  965 = 'Mc_Warnings Default 965' | German: 'Mc_Warnings German 965' | French: 'Mc_Warnings French 965'
  966 = 'Mc_Warnings Default 966' | German: 'Mc_Warnings German 966' | French: 'Mc_Warnings French 966'
  967 = 'Mc_Warnings Default 967' | German: 'Mc_Warnings German 967' | French: 'Mc_Warnings French 967'
  968 = 'Mc_Warnings Default 968' | German: 'Mc_Warnings German 968' | French: 'Mc_Warnings French 968'
  969 = 'Mc_Warnings Default 969' | German: 'Mc_Warnings German 969' | French: 'Mc_Warnings French 969'
  970 = 'Mc_Warnings Default 970' | German: 'Mc_Warnings German 970' | French: 'Mc_Warnings French 970'
  971 = 'Mc_Warnings Default 971' | German: 'Mc_Warnings German 971' | French: 'Mc_Warnings French 971'
  972 = 'Mc_Warnings Default 972' | German: 'Mc_Warnings German 972' | French: 'Mc_Warnings French 972'
  973 = 'Mc_Warnings Default 973' | German: 'Mc_Warnings German 973' | French: 'Mc_Warnings French 973'
  974 = 'Mc_Warnings Default 974' | German: 'Mc_Warnings German 974' | French: 'Mc_Warnings French 974'
  975 = 'Mc_Warnings Default 975' | German: 'Mc_Warnings German 975' | French: 'Mc_Warnings French 975'
  976 = 'Mc_Warnings Default 976' | German: 'Mc_Warnings German 976' | French: 'Mc_Warnings French 976'
  977 = 'Mc_Warnings Default 977' | German: 'Mc_Warnings German 977' | French: 'Mc_Warnings French 977'
  978 = 'Mc_Warnings Default 978' | German: 'Mc_Warnings German 978' | French: 'Mc_Warnings French 978'
  979 = 'Mc_Warnings Default 979' | German: 'Mc_Warnings German 979' | French: 'Mc_Warnings French 979'
  980 = 'Mc_Warnings Default 980' | German: 'Mc_Warnings German 980' | French: 'Mc_Warnings French 980'
  981 = 'Mc_Warnings Default 981' | German: 'Mc_Warnings German 981' | French: 'Mc_Warnings French 981'
  982 = 'Mc_Warnings Default 982' | German: 'Mc_Warnings German 982' | French: 'Mc_Warnings French 982'
  983 = 'Mc_Warnings Default 983' | German: 'Mc_Warnings German 983' | French: 'Mc_Warnings French 983'
  984 = 'Mc_Warnings Default 984' | German: 'Mc_Warnings German 984' | French: 'Mc_Warnings French 984'
  985 = 'Mc_Warnings Default 985' | German: 'Mc_Warnings German 985' | French: 'Mc_Warnings French 985'
  986 = 'Mc_Warnings Default 986' | German: 'Mc_Warnings German 986' | French: 'Mc_Warnings French 986'
  987 = 'Mc_Warnings Default 987' | German: 'Mc_Warnings German 987' | French: 'Mc_Warnings French 987'
  988 = 'Mc_Warnings Default 988' | German: 'Mc_Warnings German 988' | French: 'Mc_Warnings French 988'
  989 = 'Mc_Warnings Default 989' | German: 'Mc_Warnings German 989' | French: 'Mc_Warnings French 989'
  990 = 'Mc_Warnings Default 990' | German: 'Mc_Warnings German 990' | French: 'Mc_Warnings French 990'
  991 = 'Mc_Warnings Default 991' | German: 'Mc_Warnings German 991' | French: 'Mc_Warnings French 991'
  992 = 'Mc_Warnings Default 992' | German: 'Mc_Warnings German 992' | French: 'Mc_Warnings French 992'
  993 = 'Mc_Warnings Default 993' | German: 'Mc_Warnings German 993' | French: 'Mc_Warnings French 993'
  994 = 'Mc_Warnings Default 994' | German: 'Mc_Warnings German 994' | French: 'Mc_Warnings French 994'
  995 = 'Mc_Warnings Default 995' | German: 'Mc_Warnings German 995' | French: 'Mc_Warnings French 995'
  996 = 'Mc_Warnings Default 996' | German: 'Mc_Warnings German 996' | French: 'Mc_Warnings French 996'
  997 = 'Mc_Warnings Default 997' | German: 'Mc_Warnings German 997' | French: 'Mc_Warnings French 997'
  998 = 'Mc_Warnings Default 998' | German: 'Mc_Warnings German 998' | French: 'Mc_Warnings French 998'
  999 = 'Mc_Warnings Default 999' | German: 'Mc_Warnings German 999' | French: 'Mc_Warnings French 999'
  1000 = 'Mc_Warnings Default 1000' | German: 'Mc_Warnings German 1000' | French: 'Mc_Warnings French 1000'
   = ''
END_TEXTLIST

(* stored: Version 1.1.0.1, ProductVersion 3.1.4024.11
   TextList Mc_Warnings: Id {fd185ce1-9315-01c5-104f-3e9e22efccb8} *)
